{attribute addProperty BoxType "EK1122-0000-0018"}
{attribute addProperty Id "Beckhoff_EP5xxxsub_EK1100EK1100_179A0949162A_0001_EP5001_0002_0016EP5001_99FC62FA13016.25A_0002_EP5101_0002_0016EP5101_CA84C7C416220.25A_0003_EP5101_0002_0017EP5101_CA84C7C416220.25A_0004_EP5101_0002_0018EP5101_CA84C7C416220.25A_0005_EP5101_0002_0019EP5101_CA84C7C416220.25A_0006_EP5101_0011_0016EP5101_19FB32BA16220.25A_0007_EP5101_0011_0017EP5101_19FB32BA16220.25A_0008_EP5101_0011_0018EP5101_19FB32BA16220.25A_0009_EP5101_0011_0019EP5101_19FB32BA16220.25A_0010_EP5101_1002_0017EP5101_CA84C7C416220.25A_0011_EP5151_0002_0018EP5151_19FB32BA16220.25A_0012_EP5101_2011_0016EP5101_354B248916220.25"}
{attribute addProperty CRC "1093743672"}
{attribute addProperty SizeInBites "1928"}
{attribute addProperty SizeInBytes "241"}
TYPE Beckhoff_EP5xxxEK1122_41313438 EXTENDS EK1122_179A0949 :
STRUCT
	{attribute addProperty Name "Beckhoff_EP5xxxsub_EK1100"}
	Beckhoff_EP5xxxsub_EK1100 : EK1100_179A0949;
	{attribute addProperty Name "A_0001_EP5001_0002_0016"}
	A_0001_EP5001_0002_0016 : EP5001_99FC62FA;
	{attribute addProperty Name "A_0002_EP5101_0002_0016"}
	A_0002_EP5101_0002_0016 : EP5101_CA84C7C4;
	{attribute addProperty Name "A_0003_EP5101_0002_0017"}
	A_0003_EP5101_0002_0017 : EP5101_CA84C7C4;
	{attribute addProperty Name "A_0004_EP5101_0002_0018"}
	A_0004_EP5101_0002_0018 : EP5101_CA84C7C4;
	{attribute addProperty Name "A_0005_EP5101_0002_0019"}
	A_0005_EP5101_0002_0019 : EP5101_CA84C7C4;
	{attribute addProperty Name "A_0006_EP5101_0011_0016"}
	A_0006_EP5101_0011_0016 : EP5101_19FB32BA;
	{attribute addProperty Name "A_0007_EP5101_0011_0017"}
	A_0007_EP5101_0011_0017 : EP5101_19FB32BA;
	{attribute addProperty Name "A_0008_EP5101_0011_0018"}
	A_0008_EP5101_0011_0018 : EP5101_19FB32BA;
	{attribute addProperty Name "A_0009_EP5101_0011_0019"}
	A_0009_EP5101_0011_0019 : EP5101_19FB32BA;
	{attribute addProperty Name "A_0010_EP5101_1002_0017"}
	A_0010_EP5101_1002_0017 : EP5101_CA84C7C4;
	{attribute addProperty Name "A_0011_EP5151_0002_0018"}
	A_0011_EP5151_0002_0018 : EP5151_19FB32BA;
	{attribute addProperty Name "A_0012_EP5101_2011_0016"}
	A_0012_EP5101_2011_0016 : EP5101_354B2489;
END_STRUCT
END_TYPE

(* stored: Version 1.2.0.0, ProductVersion 3.1.4024.9
   DUT Beckhoff_EP5xxxEK1122_41313438: Id {5c7856c5-9ae1-4ddf-8188-76ffc506fd4d} *)
